FUNCTION_BLOCK FB_AxisRef_To_MSTA
VAR_INPUT
	stAxis	:	AXIS_REF;
END_VAR
VAR_OUTPUT
	MSTA	:	UINT;
END_VAR
VAR
END_VAR

(* This block translates the axis ref status to an EPICS psuedo MSTA value *)
(* A. Wallace, 17/8/17 *)

MSTA.1 := stAxis.Status.Error;
MSTA.0 := stAxis.Status.Operational;

END_FUNCTION_BLOCK

(* stored: Version 1.1.0.1, ProductVersion 3.1.4020.12
   POU FB_AxisRef_To_MSTA: Id {6037187c-3053-436d-ba08-ac7db25710cf}, SpecialFunc None *)
